{attribute 'GeneratedUsingTerminal: EL6201-0000-0017'}
{attribute addProperty BoxType "EL6201-0000-0017"}
{attribute addProperty Id "Slave_13A_DO0BOOL1Slave_13A_DO1BOOL1Slave_13A_DO2BOOL1Slave_13A_DO3BOOL1Slave_13B_DO0BOOL1Slave_13B_DO1BOOL1Slave_13B_DO2BOOL1Slave_13B_DO3BOOL1"}
{attribute addProperty CRC "2140678211"}
{attribute addProperty Size "8"}
TYPE Slave_13_Outputs_7F982843 :
STRUCT
	{attribute addProperty Name "Slave_13A_DO0"}
	Slave_13A_DO0 : BOOL;
	{attribute addProperty Name "Slave_13A_DO1"}
	Slave_13A_DO1 : BOOL;
	{attribute addProperty Name "Slave_13A_DO2"}
	Slave_13A_DO2 : BOOL;
	{attribute addProperty Name "Slave_13A_DO3"}
	Slave_13A_DO3 : BOOL;
	{attribute addProperty Name "Slave_13B_DO0"}
	Slave_13B_DO0 : BOOL;
	{attribute addProperty Name "Slave_13B_DO1"}
	Slave_13B_DO1 : BOOL;
	{attribute addProperty Name "Slave_13B_DO2"}
	Slave_13B_DO2 : BOOL;
	{attribute addProperty Name "Slave_13B_DO3"}
	Slave_13B_DO3 : BOOL;
END_STRUCT
END_TYPE

(* stored: Version 1.2.0.0, ProductVersion 3.1.4024.9
   DUT Slave_13_Outputs_7F982843: Id {d80ccfa2-c19d-4a07-8265-3342cf355842} *)
